FUNCTION_BLOCK DataPanel_xDB_16_ADI_SAE_J1939 (* Service Interface Function Block Type *)
  (* Standard: SAE J1939; Function: All Inputs; Type: DP-34044-2-000 *)
  (* Version 1.0, 2018-12-05, Jose Cabral *)
  (* Version 1.0, 2022-08-04, Franz Höpfinger, Unknown *)
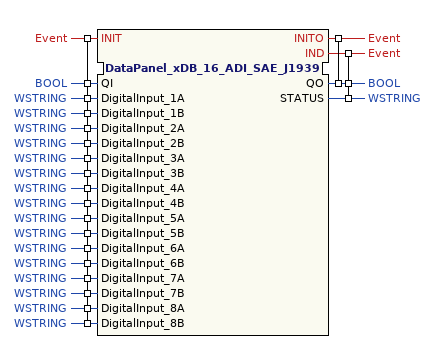
  EVENT_INPUT
    INIT WITH DigitalInput_1A, DigitalInput_1B, DigitalInput_2A, DigitalInput_2B, DigitalInput_3A, DigitalInput_3B, DigitalInput_4A, DigitalInput_4B, DigitalInput_5A, DigitalInput_5B, DigitalInput_6A, DigitalInput_6B, DigitalInput_7A, DigitalInput_7B, DigitalInput_8A, DigitalInput_8B, QI; (* Service Initialization *)
  END_EVENT
  EVENT_OUTPUT
    INITO WITH QO; (* Initialization Confirm *)
    IND WITH QO, STATUS; (* Indication from Resource *)
  END_EVENT
  VAR_INPUT
    QI : BOOL; (* Event Input Qualifier *)
    DigitalInput_1A : WSTRING;
    DigitalInput_1B : WSTRING;
    DigitalInput_2A : WSTRING;
    DigitalInput_2B : WSTRING;
    DigitalInput_3A : WSTRING;
    DigitalInput_3B : WSTRING;
    DigitalInput_4A : WSTRING;
    DigitalInput_4B : WSTRING;
    DigitalInput_5A : WSTRING;
    DigitalInput_5B : WSTRING;
    DigitalInput_6A : WSTRING;
    DigitalInput_6B : WSTRING;
    DigitalInput_7A : WSTRING;
    DigitalInput_7B : WSTRING;
    DigitalInput_8A : WSTRING;
    DigitalInput_8B : WSTRING;
  END_VAR
  VAR_OUTPUT
    QO : BOOL; (* Event Output Qualifier *)
    STATUS : WSTRING; (* Service Status *)
  END_VAR
END_FUNCTION_BLOCK
